// TIA Portal V20 export
DATA_BLOCK "SBK04"   // DB215
// stored: MemoryReserve 100
   VAR
      "X1-0 Gate EC TOP: Lock" : Bool;
      "X2-1 Gate EC TOP: Reset" : Bool;
      "X3-2 DIFFERENTIAL PRESSURE SWITCH 1 NC" : Bool;
      "X4-3 DIFFERENTIAL PRESSURE SWITCH 2 NC" : Bool;
      "X1-4 Gate EC TOP: Unlock" : Bool;
      "X2-5 reserved" : Bool;
      "X3-6 reserved" : Bool;
      "X4-7 reserved" : Bool;
      "X5-0 Gate EC TOP: Lock lamp on" : Bool;
      "X6-1 Gate EC TOP: Unlock lamp on" : Bool;
      "X7-2 Gate EC TOP: Reset lamp on" : Bool;
   END_VAR
BEGIN
END_DATA_BLOCK
